PROGRAM MAIN
VAR
END_VAR

P_Tc2DALI_KL6821();

END_PROGRAM

(* stored: Version 1.1.0.1, ProductVersion 3.1.4024.0
   POU MAIN: Id {ab8642c9-a44f-41ec-ad41-382be9b284ba}, SpecialFunc None *)
